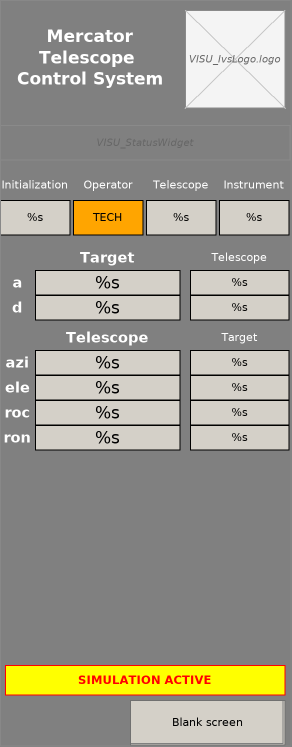
VISUALIZATION VISU_MTCSSidebar  // 292x747
VAR_IN_OUT
	mtcs : MTCS;
	mtcsWidget : MTCSWidget;
END_VAR
    Rectangle (5,25 170x65), "Mercator Telescope Control System"
    Label (0,170 70x30), "Initialization"
    Image (185,10 100x98), image: VISU_IvsLogo.logo
    Label (73,170 70x30), "Operator"
    Rectangle (73,200 70x35), "Observer", invisible if: NOT mtcs.statuses.operatorStatus.observer
        OnMouseClick: OpenDialog Dialog=VISU_MTCSChangeOperatorDialog, OpenModal=True, OpenCentered=True
    Rectangle (73,200 70x35), "TECH", invisible if: NOT mtcs.statuses.operatorStatus.tech
        OnMouseClick: OpenDialog Dialog=VISU_MTCSChangeOperatorDialog, OpenModal=True, OpenCentered=True
    Rectangle (0,200 70x35), "%s", text variable: mtcsWidget.initializationStatus.description, colour variable: mtcsWidget.initializationStatus.bgColor
        p55702900: mtcsWidget.initializationStatus.fgColor
        p3450524324: mtcsWidget.initializationStatus.fgColor
    Rectangle (5,665 280x30), "SIMULATION ACTIVE", invisible if: NOT GLOBAL.config.SIMULATION_ACTIVE
    Label (146,170 70x30), "Telescope"
    Rectangle (146,200 70x35), "%s", text variable: mtcsWidget.activityStatus.description, colour variable: mtcsWidget.activityStatus.bgColor
        p55702900: mtcsWidget.activityStatus.fgColor
        p3450524324: mtcsWidget.activityStatus.fgColor
    Rectangle (219,200 70x35), "%s", text variable: mtcsWidget.changeInstrumentStatus.text, colour variable: mtcsWidget.changeInstrumentStatus.color.bg
        p55702900: mtcsWidget.changeInstrumentStatus.color.fg
        p3450524324: mtcsWidget.changeInstrumentStatus.color.fg
    Button (130,700 155x45), "Blank screen"
        OnMouseClick: change screen: VISU_MTCSBlankScreen
    Label (219,170 70x30), "Instrument"
    Frame (0,125 290x35)
        shows VISU_StatusWidget(widget := mtcsWidget.actualStatus)
    Label (35,245 145x25), "Target"
    Label (0,270 35x25), "a"
    Label (0,295 35x25), "d"
    Label (190,245 99x25), "Telescope"
    Rectangle (35,270 145x25), "%s", text variable: mtcsWidget.axes.target.alphaString
    Rectangle (35,295 145x25), "%s", text variable: mtcsWidget.axes.target.deltaString
    Rectangle (190,270 99x25), "%s", text variable: mtcsWidget.axes.feedback.alpha.hmsString
    Rectangle (190,295 99x25), "%s", text variable: mtcsWidget.axes.feedback.delta.dmsString
    Label (35,325 145x25), "Telescope"
    Label (0,350 35x25), "azi"
    Label (190,325 99x25), "Target"
    Rectangle (35,350 145x25), "%s", text variable: mtcsWidget.axes.feedback.aziPos.dmsString
    Rectangle (190,350 99x25), "%s", text variable: mtcsWidget.axes.target.aziString
    Label (0,375 35x25), "ele"
    Rectangle (35,375 145x25), "%s", text variable: mtcsWidget.axes.feedback.elePos.dmsString
    Rectangle (190,375 99x25), "%s", text variable: mtcsWidget.axes.target.eleString
    Label (0,400 35x25), "roc"
    Rectangle (35,400 145x25), "%s", text variable: mtcsWidget.axes.feedback.rocPos.dmsString
    Rectangle (190,425 99x25), "%s", text variable: mtcsWidget.axes.target.paString
    Label (0,425 35x25), "ron"
    Rectangle (35,425 145x25), "%s", text variable: mtcsWidget.axes.feedback.ronPos.dmsString
    Rectangle (190,400 99x25), "%s", text variable: mtcsWidget.axes.target.paString
END_VISUALIZATION

(* stored: Version 1.1.0.1, ProductVersion 3.1.4019.2
   Visu VISU_MTCSSidebar: Id {36d59378-aa06-4df0-a93f-51a001c7a70e} *)
